// Mitsubishi GX Works2 project: 20150731_final8_test   PLC: Q02/Q02H

PROGRAM MAIN
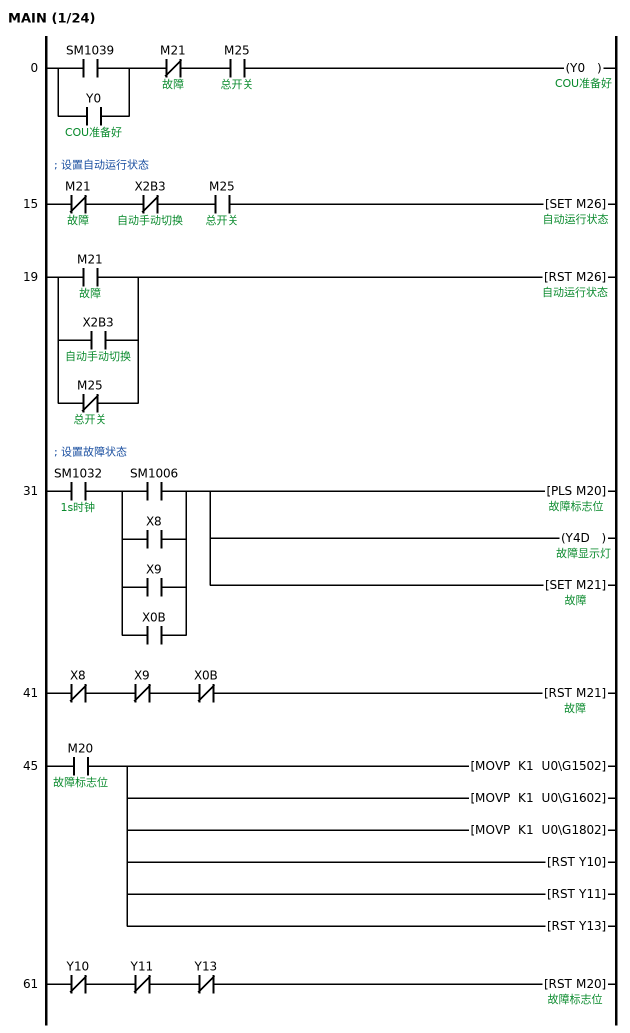
0     LD      SM1039
      OR      Y0  ; COU准备好
      ANI     M21  ; 故障
      AND     M25  ; 总开关
      OUT     Y0  ; COU准备好
; 设置自动运行状态
15    LDI     M21  ; 故障
      ANI     X2B3  ; 自动手动切换
      AND     M25  ; 总开关
      SET     M26  ; 自动运行状态
19    LD      M21  ; 故障
      OR      X2B3  ; 自动手动切换
      ORI     M25  ; 总开关
      RST     M26  ; 自动运行状态
; 设置故障状态
31    LD      SM1032  ; 1s时钟
      LD      SM1006
      OR      X8
      OR      X9
      OR      X0B
      ANB
      PLS     M20  ; 故障标志位
      OUT     Y4D  ; 故障显示灯
      SET     M21  ; 故障
41    LDI     X8
      ANI     X9
      ANI     X0B
      RST     M21  ; 故障
45    LD      M20  ; 故障标志位
      MOVP    K1 U0\G1502
      MOVP    K1 U0\G1602
      MOVP    K1 U0\G1802
      RST     Y10
      RST     Y11
      RST     Y13
61    LDI     Y10
      ANI     Y11
      ANI     Y13
      RST     M20  ; 故障标志位
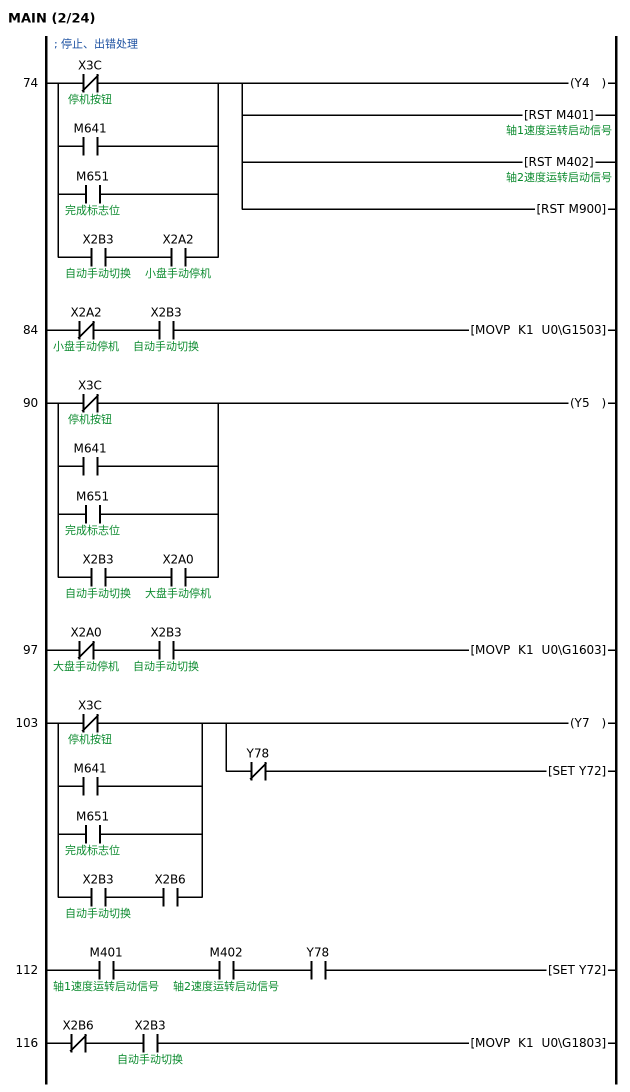
; 停止、出错处理
74    LDI     X3C  ; 停机按钮
      OR      M641
      OR      M651  ; 完成标志位
      LD      X2B3  ; 自动手动切换
      AND     X2A2  ; 小盘手动停机
      ORB
      OUT     Y4
      RST     M401  ; 轴1速度运转启动信号
      RST     M402  ; 轴2速度运转启动信号
      RST     M900
84    LDI     X2A2  ; 小盘手动停机
      AND     X2B3  ; 自动手动切换
      MOVP    K1 U0\G1503
90    LDI     X3C  ; 停机按钮
      OR      M641
      OR      M651  ; 完成标志位
      LD      X2B3  ; 自动手动切换
      AND     X2A0  ; 大盘手动停机
      ORB
      OUT     Y5
97    LDI     X2A0  ; 大盘手动停机
      AND     X2B3  ; 自动手动切换
      MOVP    K1 U0\G1603
103   LDI     X3C  ; 停机按钮
      OR      M641
      OR      M651  ; 完成标志位
      LD      X2B3  ; 自动手动切换
      AND     X2B6
      ORB
      OUT     Y7
      ANI     Y78
      SET     Y72
112   LD      M401  ; 轴1速度运转启动信号
      AND     M402  ; 轴2速度运转启动信号
      AND     Y78
      SET     Y72
116   LDI     X2B6
      AND     X2B3  ; 自动手动切换
      MOVP    K1 U0\G1803
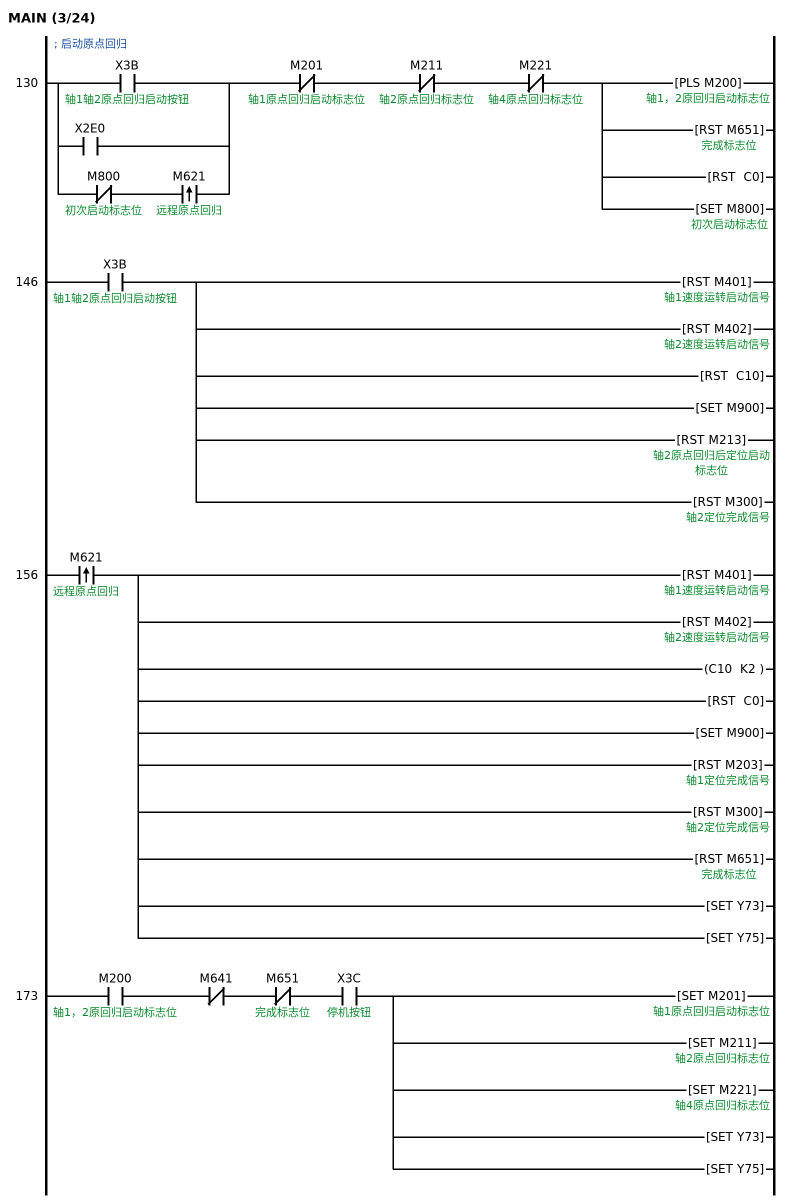
; 启动原点回归
130   LD      X3B  ; 轴1轴2原点回归启动按钮
      OR      X2E0
      LDI     M800  ; 初次启动标志位
      ANDP    M621  ; 远程原点回归
      ORB
      ANI     M201  ; 轴1原点回归启动标志位
      ANI     M211  ; 轴2原点回归标志位
      ANI     M221  ; 轴4原点回归标志位
      PLS     M200  ; 轴1，2原回归启动标志位
      RST     M651  ; 完成标志位
      RST     C0
      SET     M800  ; 初次启动标志位
146   LD      X3B  ; 轴1轴2原点回归启动按钮
      RST     M401  ; 轴1速度运转启动信号
      RST     M402  ; 轴2速度运转启动信号
      RST     C10
      SET     M900
      RST     M213  ; 轴2原点回归后定位启动标志位
      RST     M300  ; 轴2定位完成信号
156   LDP     M621  ; 远程原点回归
      RST     M401  ; 轴1速度运转启动信号
      RST     M402  ; 轴2速度运转启动信号
      OUT     C10 K2
      RST     C0
      SET     M900
      RST     M203  ; 轴1定位完成信号
      RST     M300  ; 轴2定位完成信号
      RST     M651  ; 完成标志位
      SET     Y73
      SET     Y75
173   LD      M200  ; 轴1，2原回归启动标志位
      ANI     M641
      ANI     M651  ; 完成标志位
      AND     X3C  ; 停机按钮
      SET     M201  ; 轴1原点回归启动标志位
      SET     M211  ; 轴2原点回归标志位
      SET     M221  ; 轴4原点回归标志位
      SET     Y73
      SET     Y75
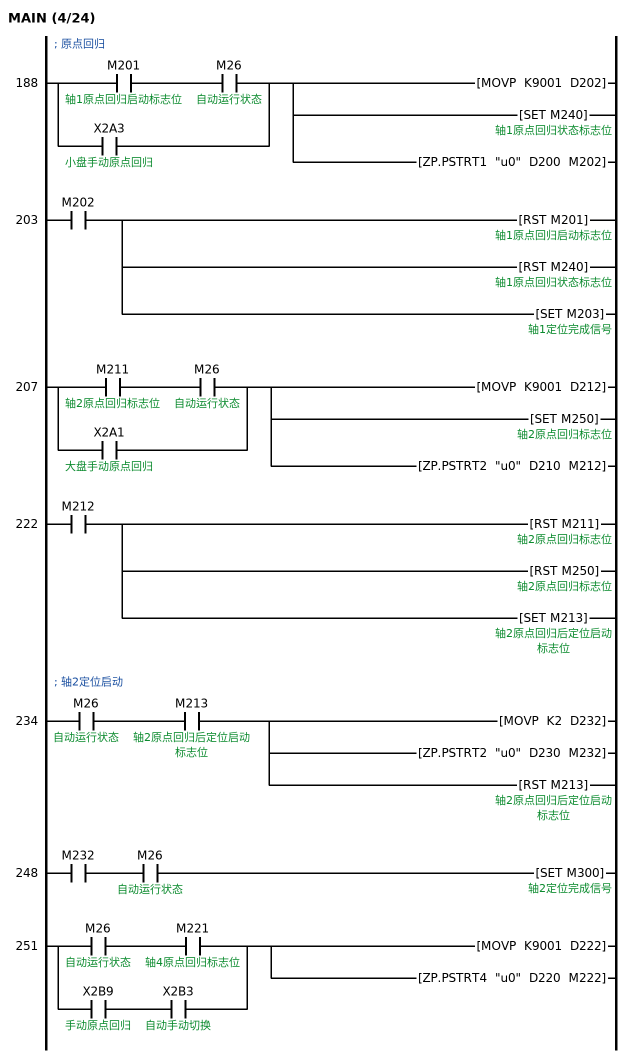
; 原点回归
188   LD      M201  ; 轴1原点回归启动标志位
      AND     M26  ; 自动运行状态
      OR      X2A3  ; 小盘手动原点回归
      MOVP    K9001 D202
      SET     M240  ; 轴1原点回归状态标志位
      ZP.PSTRT1 "u0" D200 M202
203   LD      M202
      RST     M201  ; 轴1原点回归启动标志位
      RST     M240  ; 轴1原点回归状态标志位
      SET     M203  ; 轴1定位完成信号
207   LD      M211  ; 轴2原点回归标志位
      AND     M26  ; 自动运行状态
      OR      X2A1  ; 大盘手动原点回归
      MOVP    K9001 D212
      SET     M250  ; 轴2原点回归标志位
      ZP.PSTRT2 "u0" D210 M212
222   LD      M212
      RST     M211  ; 轴2原点回归标志位
      RST     M250  ; 轴2原点回归标志位
      SET     M213  ; 轴2原点回归后定位启动标志位
; 轴2定位启动
234   LD      M26  ; 自动运行状态
      AND     M213  ; 轴2原点回归后定位启动标志位
      MOVP    K2 D232
      ZP.PSTRT2 "u0" D230 M232
      RST     M213  ; 轴2原点回归后定位启动标志位
248   LD      M232
      AND     M26  ; 自动运行状态
      SET     M300  ; 轴2定位完成信号
251   LD      M26  ; 自动运行状态
      AND     M221  ; 轴4原点回归标志位
      LD      X2B9  ; 手动原点回归
      AND     X2B3  ; 自动手动切换
      ORB
      MOVP    K9001 D222
      ZP.PSTRT4 "u0" D220 M222
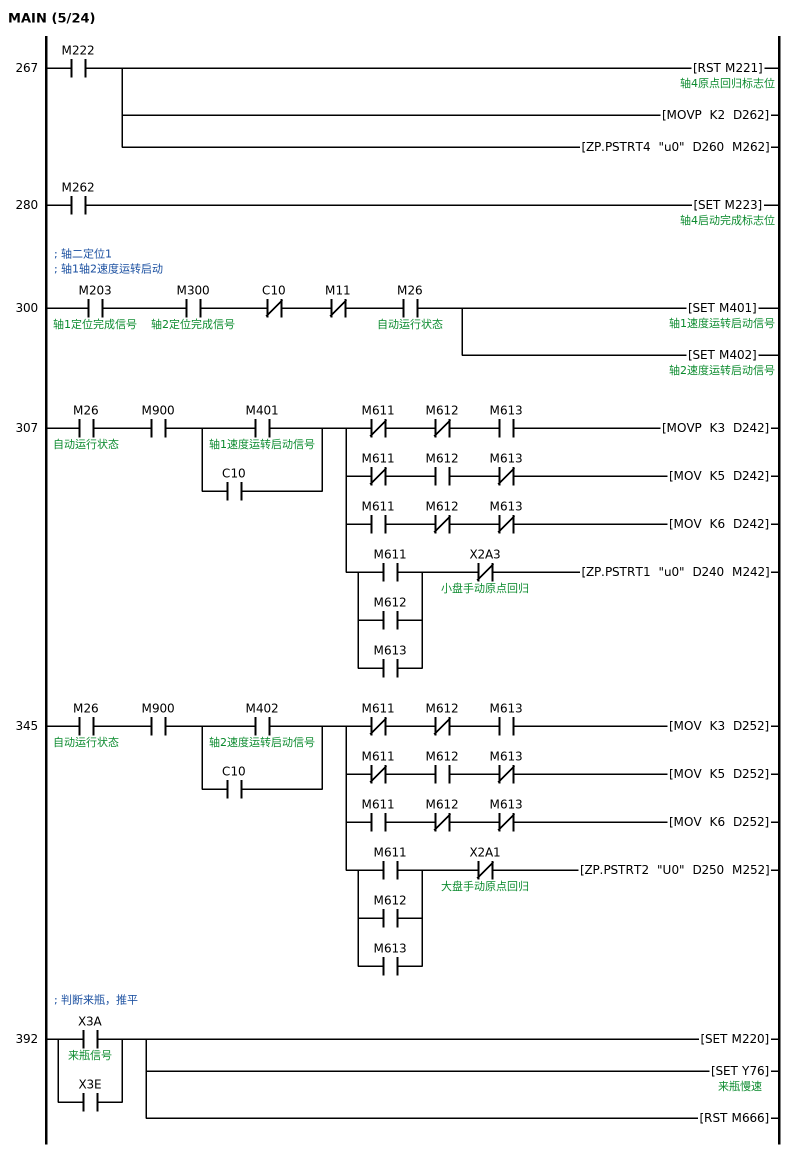
267   LD      M222
      RST     M221  ; 轴4原点回归标志位
      MOVP    K2 D262
      ZP.PSTRT4 "u0" D260 M262
280   LD      M262
      SET     M223  ; 轴4启动完成标志位
; 轴二定位1
; 轴1轴2速度运转启动
300   LD      M203  ; 轴1定位完成信号
      AND     M300  ; 轴2定位完成信号
      ANI     C10
      ANI     M11
      AND     M26  ; 自动运行状态
      SET     M401  ; 轴1速度运转启动信号
      SET     M402  ; 轴2速度运转启动信号
307   LD      M26  ; 自动运行状态
      AND     M900
      LD      M401  ; 轴1速度运转启动信号
      OR      C10
      ANB
      MPS
      ANI     M611
      ANI     M612
      AND     M613
      MOVP    K3 D242
      MRD
      ANI     M611
      AND     M612
      ANI     M613
      MOV     K5 D242
      MRD
      AND     M611
      ANI     M612
      ANI     M613
      MOV     K6 D242
      MPP
      LD      M611
      OR      M612
      OR      M613
      ANB
      ANI     X2A3  ; 小盘手动原点回归
      ZP.PSTRT1 "u0" D240 M242
345   LD      M26  ; 自动运行状态
      AND     M900
      LD      M402  ; 轴2速度运转启动信号
      OR      C10
      ANB
      MPS
      ANI     M611
      ANI     M612
      AND     M613
      MOV     K3 D252
      MRD
      ANI     M611
      AND     M612
      ANI     M613
      MOV     K5 D252
      MRD
      AND     M611
      ANI     M612
      ANI     M613
      MOV     K6 D252
      MPP
      LD      M611
      OR      M612
      OR      M613
      ANB
      ANI     X2A1  ; 大盘手动原点回归
      ZP.PSTRT2 "U0" D250 M252
; 判断来瓶，推平
392   LD      X3A  ; 来瓶信号
      OR      X3E
      SET     M220
      SET     Y76  ; 来瓶慢速
      RST     M666
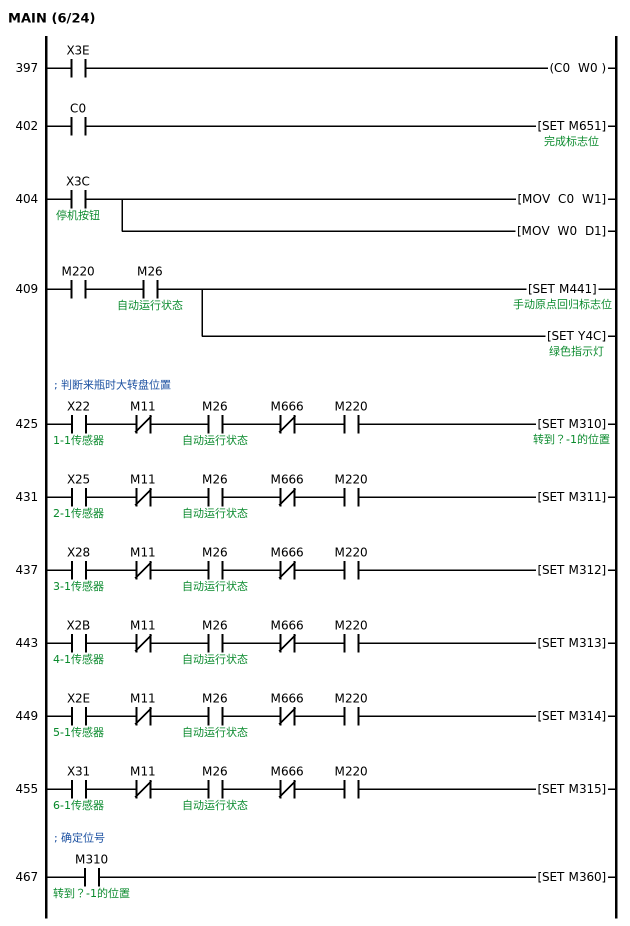
397   LD      X3E
      OUT     C0 W0
402   LD      C0
      SET     M651  ; 完成标志位
404   LD      X3C  ; 停机按钮
      MOV     C0 W1
      MOV     W0 D1
409   LD      M220
      AND     M26  ; 自动运行状态
      SET     M441  ; 手动原点回归标志位
      SET     Y4C  ; 绿色指示灯
; 判断来瓶时大转盘位置
425   LD      X22  ; 1-1传感器
      ANI     M11
      AND     M26  ; 自动运行状态
      ANI     M666
      AND     M220
      SET     M310  ; 转到？-1的位置
431   LD      X25  ; 2-1传感器
      ANI     M11
      AND     M26  ; 自动运行状态
      ANI     M666
      AND     M220
      SET     M311
437   LD      X28  ; 3-1传感器
      ANI     M11
      AND     M26  ; 自动运行状态
      ANI     M666
      AND     M220
      SET     M312
443   LD      X2B  ; 4-1传感器
      ANI     M11
      AND     M26  ; 自动运行状态
      ANI     M666
      AND     M220
      SET     M313
449   LD      X2E  ; 5-1传感器
      ANI     M11
      AND     M26  ; 自动运行状态
      ANI     M666
      AND     M220
      SET     M314
455   LD      X31  ; 6-1传感器
      ANI     M11
      AND     M26  ; 自动运行状态
      ANI     M666
      AND     M220
      SET     M315
; 确定位号
467   LD      M310  ; 转到？-1的位置
      SET     M360
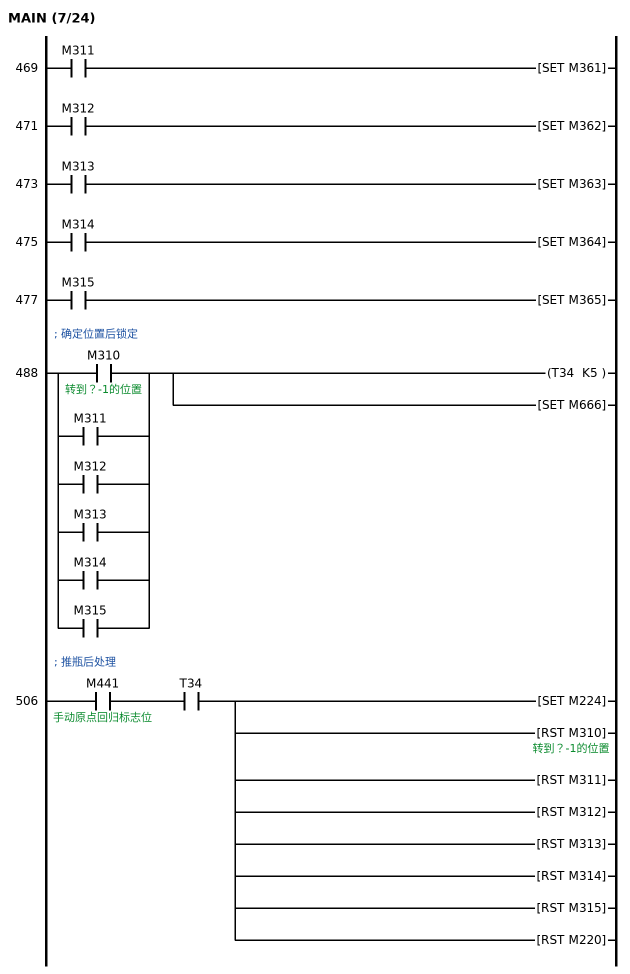
469   LD      M311
      SET     M361
471   LD      M312
      SET     M362
473   LD      M313
      SET     M363
475   LD      M314
      SET     M364
477   LD      M315
      SET     M365
; 确定位置后锁定
488   LD      M310  ; 转到？-1的位置
      OR      M311
      OR      M312
      OR      M313
      OR      M314
      OR      M315
      OUT     T34 K5
      SET     M666
; 推瓶后处理
506   LD      M441  ; 手动原点回归标志位
      AND     T34
      SET     M224
      RST     M310  ; 转到？-1的位置
      RST     M311
      RST     M312
      RST     M313
      RST     M314
      RST     M315
      RST     M220
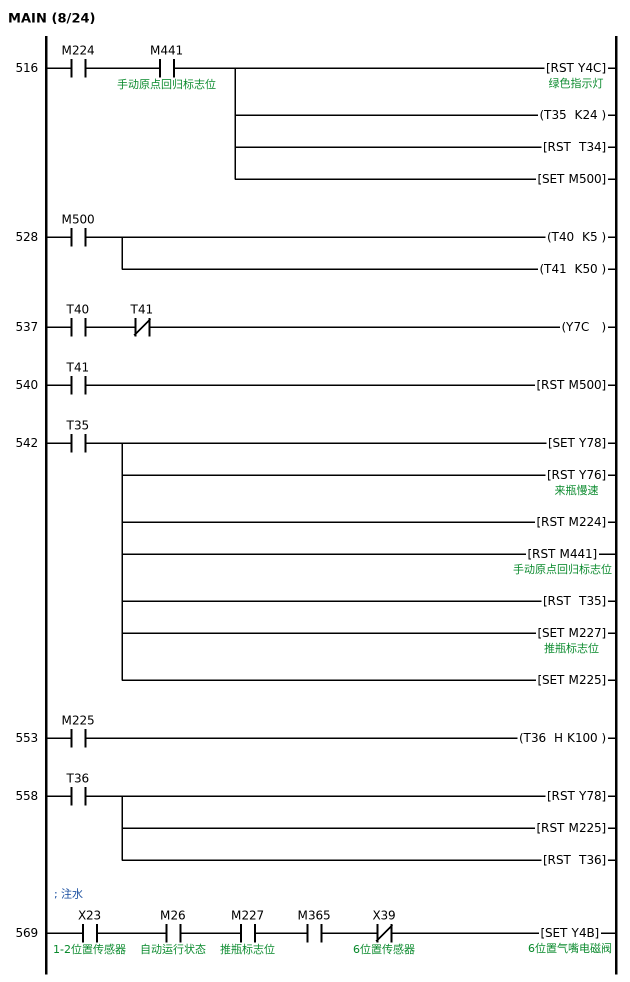
516   LD      M224
      AND     M441  ; 手动原点回归标志位
      RST     Y4C  ; 绿色指示灯
      OUT     T35 K24
      RST     T34
      SET     M500
528   LD      M500
      OUT     T40 K5
      OUT     T41 K50
537   LD      T40
      ANI     T41
      OUT     Y7C
540   LD      T41
      RST     M500
542   LD      T35
      SET     Y78
      RST     Y76  ; 来瓶慢速
      RST     M224
      RST     M441  ; 手动原点回归标志位
      RST     T35
      SET     M227  ; 推瓶标志位
      SET     M225
553   LD      M225
      OUTH    T36 K100
558   LD      T36
      RST     Y78
      RST     M225
      RST     T36
; 注水
569   LD      X23  ; 1-2位置传感器
      AND     M26  ; 自动运行状态
      AND     M227  ; 推瓶标志位
      AND     M365
      ANI     X39  ; 6位置传感器
      SET     Y4B  ; 6位置气嘴电磁阀
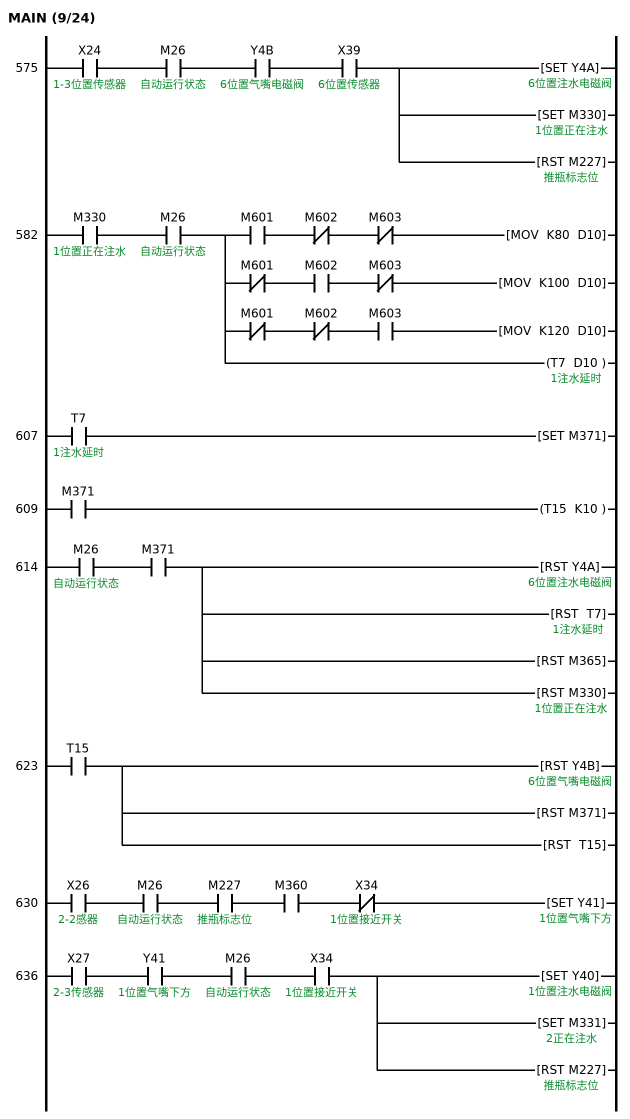
575   LD      X24  ; 1-3位置传感器
      AND     M26  ; 自动运行状态
      AND     Y4B  ; 6位置气嘴电磁阀
      AND     X39  ; 6位置传感器
      SET     Y4A  ; 6位置注水电磁阀
      SET     M330  ; 1位置正在注水
      RST     M227  ; 推瓶标志位
582   LD      M330  ; 1位置正在注水
      AND     M26  ; 自动运行状态
      MPS
      AND     M601
      ANI     M602
      ANI     M603
      MOV     K80 D10
      MRD
      ANI     M601
      AND     M602
      ANI     M603
      MOV     K100 D10
      MRD
      ANI     M601
      ANI     M602
      AND     M603
      MOV     K120 D10
      MPP
      OUT     T7 D10  ; 1注水延时
607   LD      T7  ; 1注水延时
      SET     M371
609   LD      M371
      OUT     T15 K10
614   LD      M26  ; 自动运行状态
      AND     M371
      RST     Y4A  ; 6位置注水电磁阀
      RST     T7  ; 1注水延时
      RST     M365
      RST     M330  ; 1位置正在注水
623   LD      T15
      RST     Y4B  ; 6位置气嘴电磁阀
      RST     M371
      RST     T15
630   LD      X26  ; 2-2感器
      AND     M26  ; 自动运行状态
      AND     M227  ; 推瓶标志位
      AND     M360
      ANI     X34  ; 1位置接近开关
      SET     Y41  ; 1位置气嘴下方
636   LD      X27  ; 2-3传感器
      AND     Y41  ; 1位置气嘴下方
      AND     M26  ; 自动运行状态
      AND     X34  ; 1位置接近开关
      SET     Y40  ; 1位置注水电磁阀
      SET     M331  ; 2正在注水
      RST     M227  ; 推瓶标志位
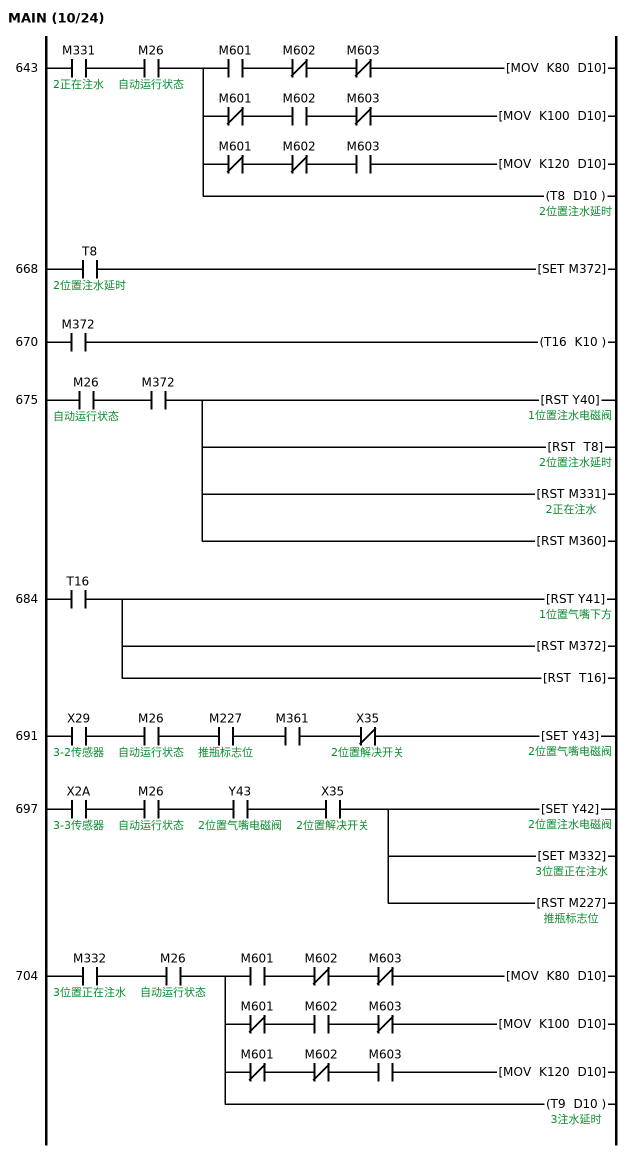
643   LD      M331  ; 2正在注水
      AND     M26  ; 自动运行状态
      MPS
      AND     M601
      ANI     M602
      ANI     M603
      MOV     K80 D10
      MRD
      ANI     M601
      AND     M602
      ANI     M603
      MOV     K100 D10
      MRD
      ANI     M601
      ANI     M602
      AND     M603
      MOV     K120 D10
      MPP
      OUT     T8 D10  ; 2位置注水延时
668   LD      T8  ; 2位置注水延时
      SET     M372
670   LD      M372
      OUT     T16 K10
675   LD      M26  ; 自动运行状态
      AND     M372
      RST     Y40  ; 1位置注水电磁阀
      RST     T8  ; 2位置注水延时
      RST     M331  ; 2正在注水
      RST     M360
684   LD      T16
      RST     Y41  ; 1位置气嘴下方
      RST     M372
      RST     T16
691   LD      X29  ; 3-2传感器
      AND     M26  ; 自动运行状态
      AND     M227  ; 推瓶标志位
      AND     M361
      ANI     X35  ; 2位置解决开关
      SET     Y43  ; 2位置气嘴电磁阀
697   LD      X2A  ; 3-3传感器
      AND     M26  ; 自动运行状态
      AND     Y43  ; 2位置气嘴电磁阀
      AND     X35  ; 2位置解决开关
      SET     Y42  ; 2位置注水电磁阀
      SET     M332  ; 3位置正在注水
      RST     M227  ; 推瓶标志位
704   LD      M332  ; 3位置正在注水
      AND     M26  ; 自动运行状态
      MPS
      AND     M601
      ANI     M602
      ANI     M603
      MOV     K80 D10
      MRD
      ANI     M601
      AND     M602
      ANI     M603
      MOV     K100 D10
      MRD
      ANI     M601
      ANI     M602
      AND     M603
      MOV     K120 D10
      MPP
      OUT     T9 D10  ; 3注水延时
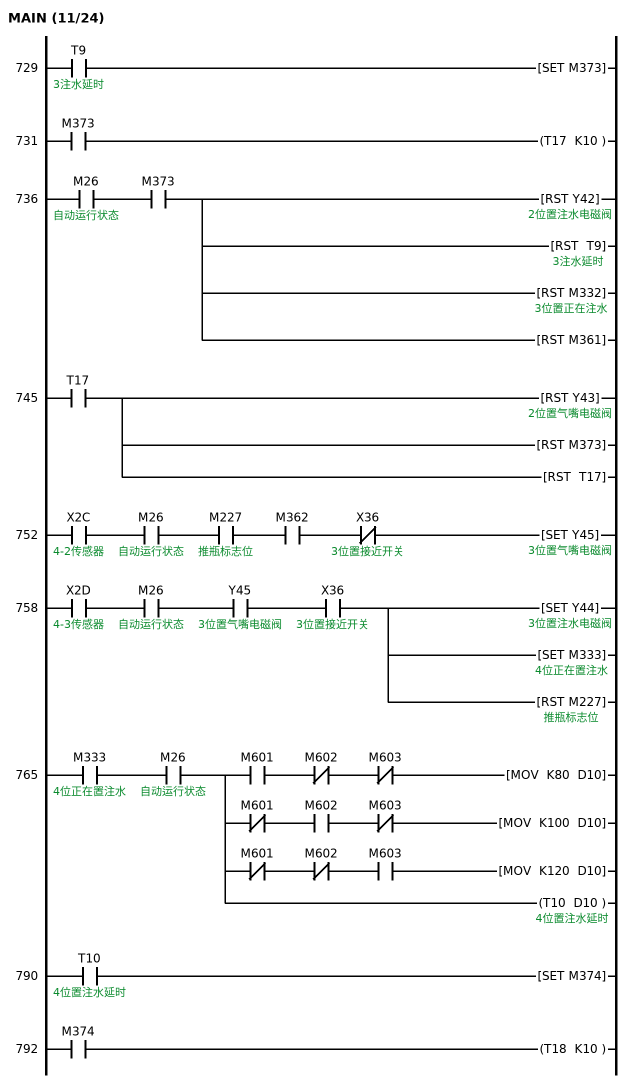
729   LD      T9  ; 3注水延时
      SET     M373
731   LD      M373
      OUT     T17 K10
736   LD      M26  ; 自动运行状态
      AND     M373
      RST     Y42  ; 2位置注水电磁阀
      RST     T9  ; 3注水延时
      RST     M332  ; 3位置正在注水
      RST     M361
745   LD      T17
      RST     Y43  ; 2位置气嘴电磁阀
      RST     M373
      RST     T17
752   LD      X2C  ; 4-2传感器
      AND     M26  ; 自动运行状态
      AND     M227  ; 推瓶标志位
      AND     M362
      ANI     X36  ; 3位置接近开关
      SET     Y45  ; 3位置气嘴电磁阀
758   LD      X2D  ; 4-3传感器
      AND     M26  ; 自动运行状态
      AND     Y45  ; 3位置气嘴电磁阀
      AND     X36  ; 3位置接近开关
      SET     Y44  ; 3位置注水电磁阀
      SET     M333  ; 4位正在置注水
      RST     M227  ; 推瓶标志位
765   LD      M333  ; 4位正在置注水
      AND     M26  ; 自动运行状态
      MPS
      AND     M601
      ANI     M602
      ANI     M603
      MOV     K80 D10
      MRD
      ANI     M601
      AND     M602
      ANI     M603
      MOV     K100 D10
      MRD
      ANI     M601
      ANI     M602
      AND     M603
      MOV     K120 D10
      MPP
      OUT     T10 D10  ; 4位置注水延时
790   LD      T10  ; 4位置注水延时
      SET     M374
792   LD      M374
      OUT     T18 K10
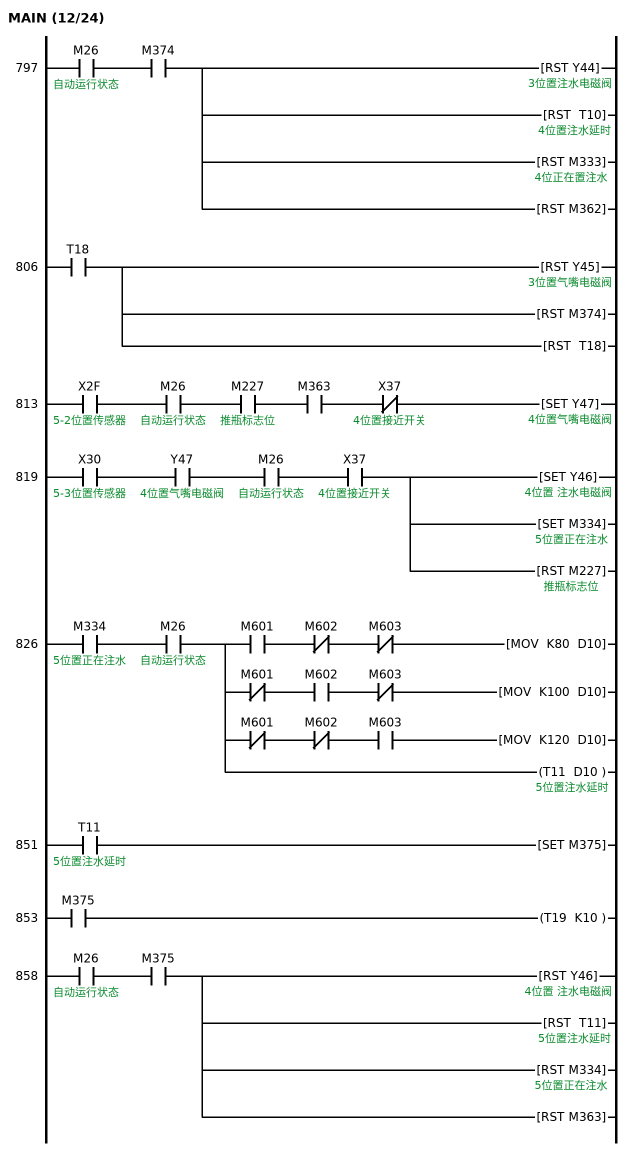
797   LD      M26  ; 自动运行状态
      AND     M374
      RST     Y44  ; 3位置注水电磁阀
      RST     T10  ; 4位置注水延时
      RST     M333  ; 4位正在置注水
      RST     M362
806   LD      T18
      RST     Y45  ; 3位置气嘴电磁阀
      RST     M374
      RST     T18
813   LD      X2F  ; 5-2位置传感器
      AND     M26  ; 自动运行状态
      AND     M227  ; 推瓶标志位
      AND     M363
      ANI     X37  ; 4位置接近开关
      SET     Y47  ; 4位置气嘴电磁阀
819   LD      X30  ; 5-3位置传感器
      AND     Y47  ; 4位置气嘴电磁阀
      AND     M26  ; 自动运行状态
      AND     X37  ; 4位置接近开关
      SET     Y46  ; 4位置 注水电磁阀
      SET     M334  ; 5位置正在注水
      RST     M227  ; 推瓶标志位
826   LD      M334  ; 5位置正在注水
      AND     M26  ; 自动运行状态
      MPS
      AND     M601
      ANI     M602
      ANI     M603
      MOV     K80 D10
      MRD
      ANI     M601
      AND     M602
      ANI     M603
      MOV     K100 D10
      MRD
      ANI     M601
      ANI     M602
      AND     M603
      MOV     K120 D10
      MPP
      OUT     T11 D10  ; 5位置注水延时
851   LD      T11  ; 5位置注水延时
      SET     M375
853   LD      M375
      OUT     T19 K10
858   LD      M26  ; 自动运行状态
      AND     M375
      RST     Y46  ; 4位置 注水电磁阀
      RST     T11  ; 5位置注水延时
      RST     M334  ; 5位置正在注水
      RST     M363
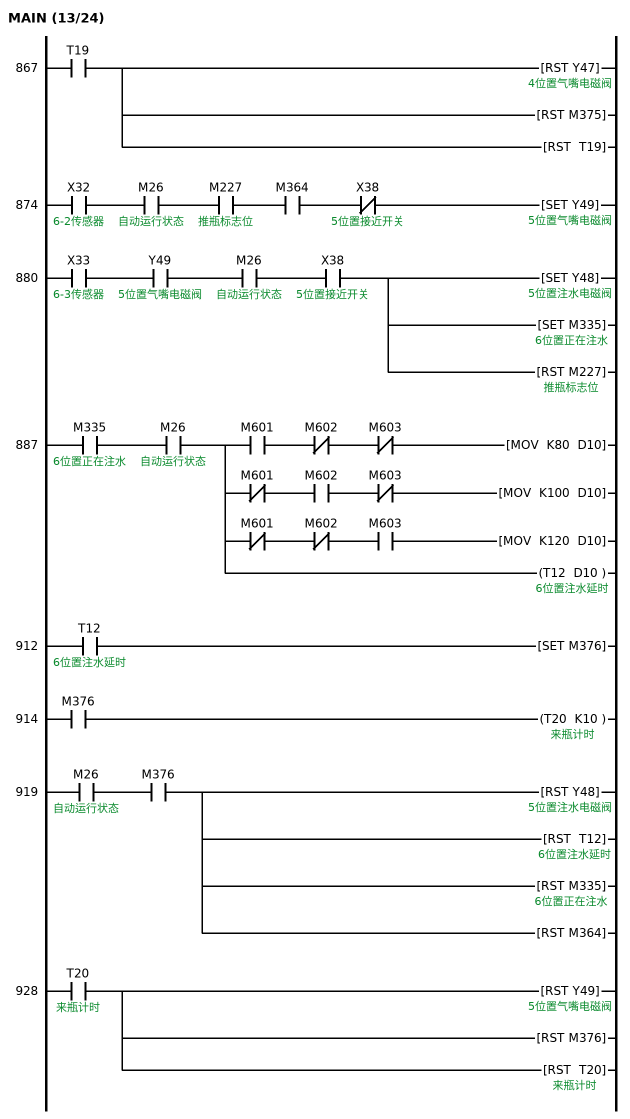
867   LD      T19
      RST     Y47  ; 4位置气嘴电磁阀
      RST     M375
      RST     T19
874   LD      X32  ; 6-2传感器
      AND     M26  ; 自动运行状态
      AND     M227  ; 推瓶标志位
      AND     M364
      ANI     X38  ; 5位置接近开关
      SET     Y49  ; 5位置气嘴电磁阀
880   LD      X33  ; 6-3传感器
      AND     Y49  ; 5位置气嘴电磁阀
      AND     M26  ; 自动运行状态
      AND     X38  ; 5位置接近开关
      SET     Y48  ; 5位置注水电磁阀
      SET     M335  ; 6位置正在注水
      RST     M227  ; 推瓶标志位
887   LD      M335  ; 6位置正在注水
      AND     M26  ; 自动运行状态
      MPS
      AND     M601
      ANI     M602
      ANI     M603
      MOV     K80 D10
      MRD
      ANI     M601
      AND     M602
      ANI     M603
      MOV     K100 D10
      MRD
      ANI     M601
      ANI     M602
      AND     M603
      MOV     K120 D10
      MPP
      OUT     T12 D10  ; 6位置注水延时
912   LD      T12  ; 6位置注水延时
      SET     M376
914   LD      M376
      OUT     T20 K10  ; 来瓶计时
919   LD      M26  ; 自动运行状态
      AND     M376
      RST     Y48  ; 5位置注水电磁阀
      RST     T12  ; 6位置注水延时
      RST     M335  ; 6位置正在注水
      RST     M364
928   LD      T20  ; 来瓶计时
      RST     Y49  ; 5位置气嘴电磁阀
      RST     M376
      RST     T20  ; 来瓶计时
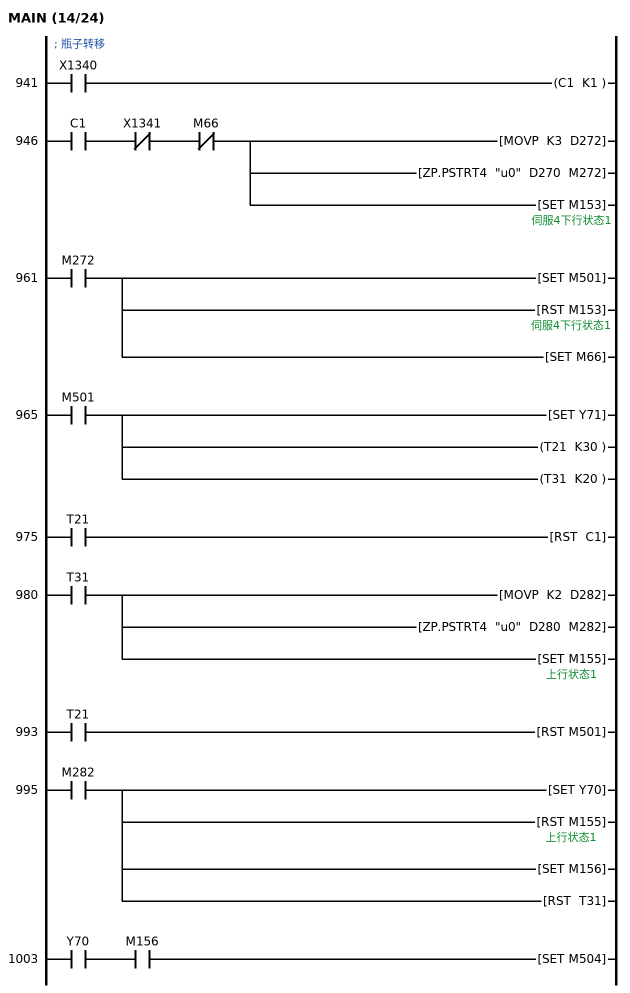
; 瓶子转移
941   LD      X1340
      OUT     C1 K1
946   LD      C1
      ANI     X1341
      ANI     M66
      MOVP    K3 D272
      ZP.PSTRT4 "u0" D270 M272
      SET     M153  ; 伺服4下行状态1
961   LD      M272
      SET     M501
      RST     M153  ; 伺服4下行状态1
      SET     M66
965   LD      M501
      SET     Y71
      OUT     T21 K30
      OUT     T31 K20
975   LD      T21
      RST     C1
980   LD      T31
      MOVP    K2 D282
      ZP.PSTRT4 "u0" D280 M282
      SET     M155  ; 上行状态1
993   LD      T21
      RST     M501
995   LD      M282
      SET     Y70
      RST     M155  ; 上行状态1
      SET     M156
      RST     T31
1003  LD      Y70
      AND     M156
      SET     M504
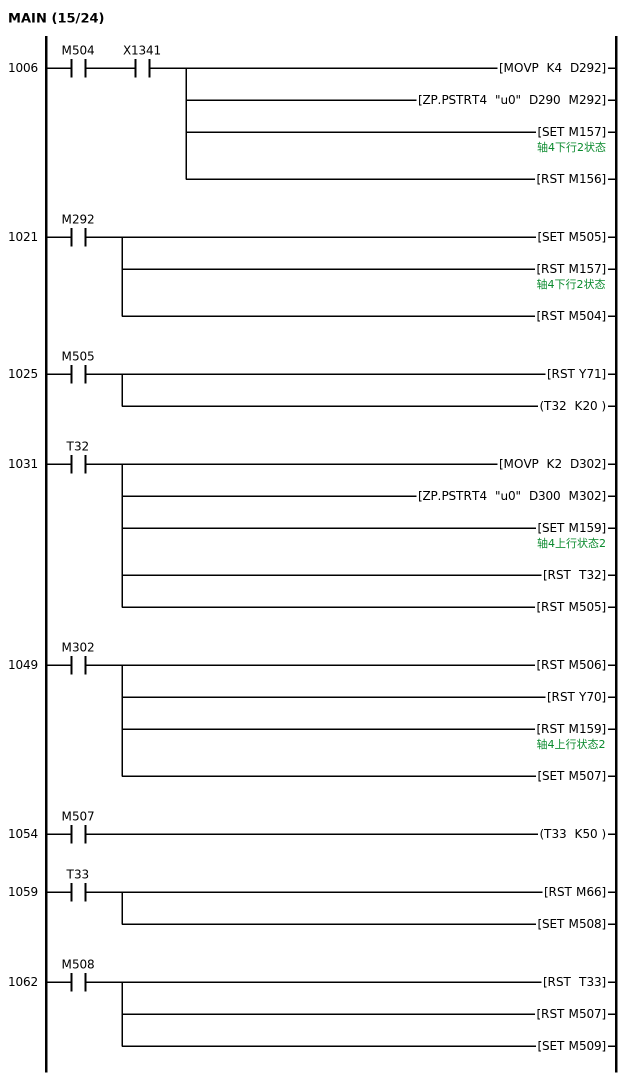
1006  LD      M504
      AND     X1341
      MOVP    K4 D292
      ZP.PSTRT4 "u0" D290 M292
      SET     M157  ; 轴4下行2状态
      RST     M156
1021  LD      M292
      SET     M505
      RST     M157  ; 轴4下行2状态
      RST     M504
1025  LD      M505
      RST     Y71
      OUT     T32 K20
1031  LD      T32
      MOVP    K2 D302
      ZP.PSTRT4 "u0" D300 M302
      SET     M159  ; 轴4上行状态2
      RST     T32
      RST     M505
1049  LD      M302
      RST     M506
      RST     Y70
      RST     M159  ; 轴4上行状态2
      SET     M507
1054  LD      M507
      OUT     T33 K50
1059  LD      T33
      RST     M66
      SET     M508
1062  LD      M508
      RST     T33
      RST     M507
      SET     M509
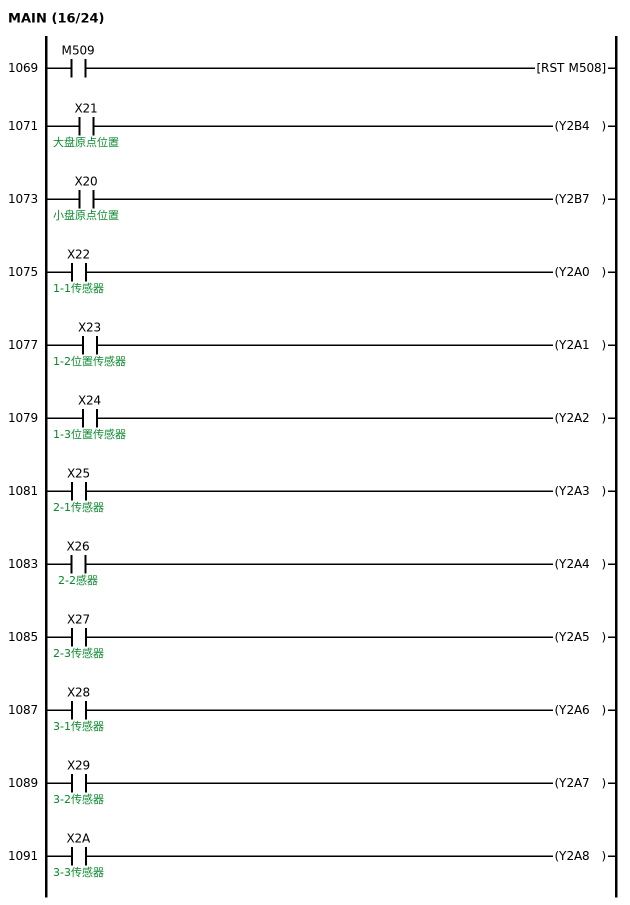
1069  LD      M509
      RST     M508
1071  LD      X21  ; 大盘原点位置
      OUT     Y2B4
1073  LD      X20  ; 小盘原点位置
      OUT     Y2B7
1075  LD      X22  ; 1-1传感器
      OUT     Y2A0
1077  LD      X23  ; 1-2位置传感器
      OUT     Y2A1
1079  LD      X24  ; 1-3位置传感器
      OUT     Y2A2
1081  LD      X25  ; 2-1传感器
      OUT     Y2A3
1083  LD      X26  ; 2-2感器
      OUT     Y2A4
1085  LD      X27  ; 2-3传感器
      OUT     Y2A5
1087  LD      X28  ; 3-1传感器
      OUT     Y2A6
1089  LD      X29  ; 3-2传感器
      OUT     Y2A7
1091  LD      X2A  ; 3-3传感器
      OUT     Y2A8
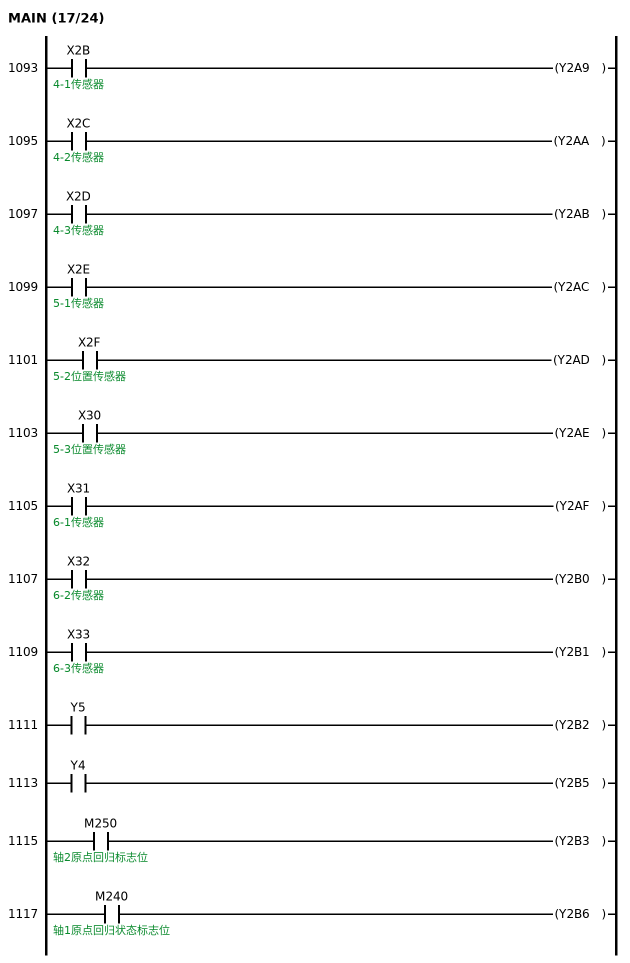
1093  LD      X2B  ; 4-1传感器
      OUT     Y2A9
1095  LD      X2C  ; 4-2传感器
      OUT     Y2AA
1097  LD      X2D  ; 4-3传感器
      OUT     Y2AB
1099  LD      X2E  ; 5-1传感器
      OUT     Y2AC
1101  LD      X2F  ; 5-2位置传感器
      OUT     Y2AD
1103  LD      X30  ; 5-3位置传感器
      OUT     Y2AE
1105  LD      X31  ; 6-1传感器
      OUT     Y2AF
1107  LD      X32  ; 6-2传感器
      OUT     Y2B0
1109  LD      X33  ; 6-3传感器
      OUT     Y2B1
1111  LD      Y5
      OUT     Y2B2
1113  LD      Y4
      OUT     Y2B5
1115  LD      M250  ; 轴2原点回归标志位
      OUT     Y2B3
1117  LD      M240  ; 轴1原点回归状态标志位
      OUT     Y2B6
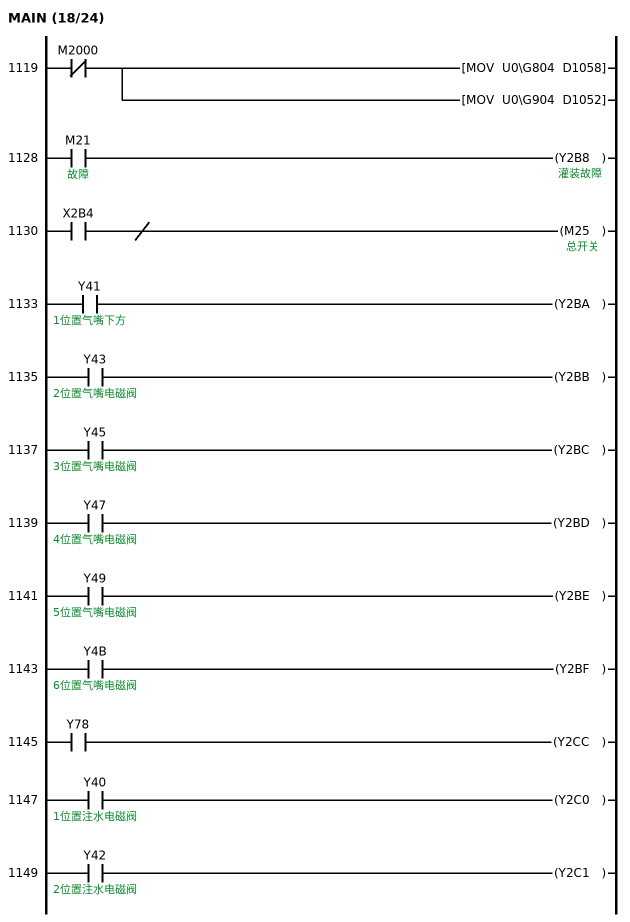
1119  LDI     M2000
      MOV     U0\G804 D1058
      MOV     U0\G904 D1052
1128  LD      M21  ; 故障
      OUT     Y2B8  ; 灌装故障
1130  LD      X2B4
      INV
      OUT     M25  ; 总开关
1133  LD      Y41  ; 1位置气嘴下方
      OUT     Y2BA
1135  LD      Y43  ; 2位置气嘴电磁阀
      OUT     Y2BB
1137  LD      Y45  ; 3位置气嘴电磁阀
      OUT     Y2BC
1139  LD      Y47  ; 4位置气嘴电磁阀
      OUT     Y2BD
1141  LD      Y49  ; 5位置气嘴电磁阀
      OUT     Y2BE
1143  LD      Y4B  ; 6位置气嘴电磁阀
      OUT     Y2BF
1145  LD      Y78
      OUT     Y2CC
1147  LD      Y40  ; 1位置注水电磁阀
      OUT     Y2C0
1149  LD      Y42  ; 2位置注水电磁阀
      OUT     Y2C1
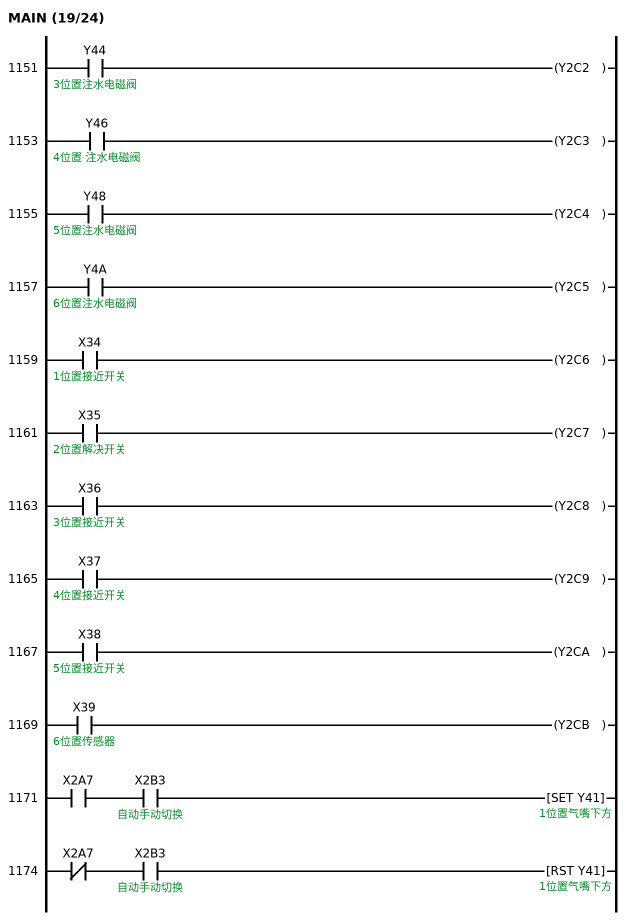
1151  LD      Y44  ; 3位置注水电磁阀
      OUT     Y2C2
1153  LD      Y46  ; 4位置 注水电磁阀
      OUT     Y2C3
1155  LD      Y48  ; 5位置注水电磁阀
      OUT     Y2C4
1157  LD      Y4A  ; 6位置注水电磁阀
      OUT     Y2C5
1159  LD      X34  ; 1位置接近开关
      OUT     Y2C6
1161  LD      X35  ; 2位置解决开关
      OUT     Y2C7
1163  LD      X36  ; 3位置接近开关
      OUT     Y2C8
1165  LD      X37  ; 4位置接近开关
      OUT     Y2C9
1167  LD      X38  ; 5位置接近开关
      OUT     Y2CA
1169  LD      X39  ; 6位置传感器
      OUT     Y2CB
1171  LD      X2A7
      AND     X2B3  ; 自动手动切换
      SET     Y41  ; 1位置气嘴下方
1174  LDI     X2A7
      AND     X2B3  ; 自动手动切换
      RST     Y41  ; 1位置气嘴下方
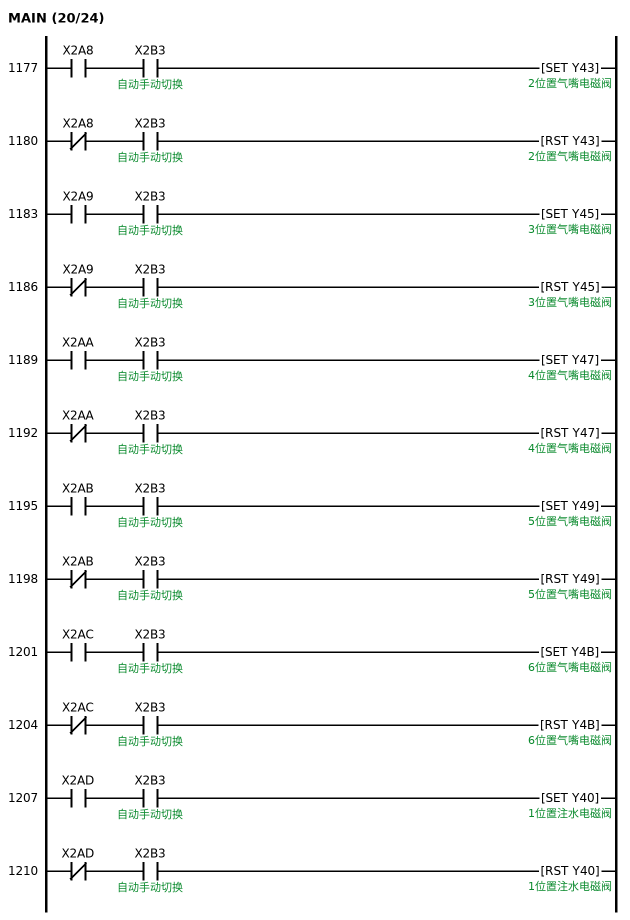
1177  LD      X2A8
      AND     X2B3  ; 自动手动切换
      SET     Y43  ; 2位置气嘴电磁阀
1180  LDI     X2A8
      AND     X2B3  ; 自动手动切换
      RST     Y43  ; 2位置气嘴电磁阀
1183  LD      X2A9
      AND     X2B3  ; 自动手动切换
      SET     Y45  ; 3位置气嘴电磁阀
1186  LDI     X2A9
      AND     X2B3  ; 自动手动切换
      RST     Y45  ; 3位置气嘴电磁阀
1189  LD      X2AA
      AND     X2B3  ; 自动手动切换
      SET     Y47  ; 4位置气嘴电磁阀
1192  LDI     X2AA
      AND     X2B3  ; 自动手动切换
      RST     Y47  ; 4位置气嘴电磁阀
1195  LD      X2AB
      AND     X2B3  ; 自动手动切换
      SET     Y49  ; 5位置气嘴电磁阀
1198  LDI     X2AB
      AND     X2B3  ; 自动手动切换
      RST     Y49  ; 5位置气嘴电磁阀
1201  LD      X2AC
      AND     X2B3  ; 自动手动切换
      SET     Y4B  ; 6位置气嘴电磁阀
1204  LDI     X2AC
      AND     X2B3  ; 自动手动切换
      RST     Y4B  ; 6位置气嘴电磁阀
1207  LD      X2AD
      AND     X2B3  ; 自动手动切换
      SET     Y40  ; 1位置注水电磁阀
1210  LDI     X2AD
      AND     X2B3  ; 自动手动切换
      RST     Y40  ; 1位置注水电磁阀
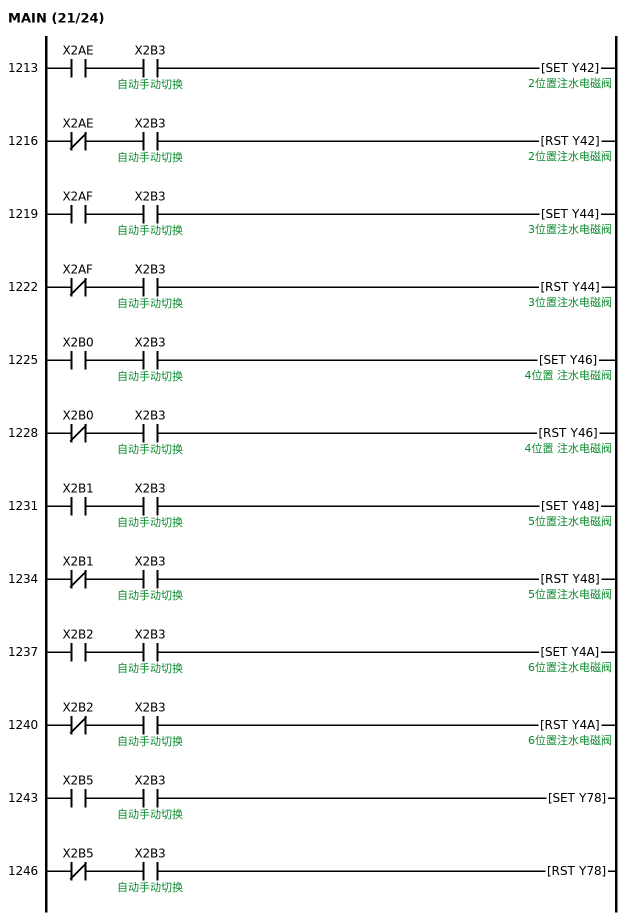
1213  LD      X2AE
      AND     X2B3  ; 自动手动切换
      SET     Y42  ; 2位置注水电磁阀
1216  LDI     X2AE
      AND     X2B3  ; 自动手动切换
      RST     Y42  ; 2位置注水电磁阀
1219  LD      X2AF
      AND     X2B3  ; 自动手动切换
      SET     Y44  ; 3位置注水电磁阀
1222  LDI     X2AF
      AND     X2B3  ; 自动手动切换
      RST     Y44  ; 3位置注水电磁阀
1225  LD      X2B0
      AND     X2B3  ; 自动手动切换
      SET     Y46  ; 4位置 注水电磁阀
1228  LDI     X2B0
      AND     X2B3  ; 自动手动切换
      RST     Y46  ; 4位置 注水电磁阀
1231  LD      X2B1
      AND     X2B3  ; 自动手动切换
      SET     Y48  ; 5位置注水电磁阀
1234  LDI     X2B1
      AND     X2B3  ; 自动手动切换
      RST     Y48  ; 5位置注水电磁阀
1237  LD      X2B2
      AND     X2B3  ; 自动手动切换
      SET     Y4A  ; 6位置注水电磁阀
1240  LDI     X2B2
      AND     X2B3  ; 自动手动切换
      RST     Y4A  ; 6位置注水电磁阀
1243  LD      X2B5
      AND     X2B3  ; 自动手动切换
      SET     Y78
1246  LDI     X2B5
      AND     X2B3  ; 自动手动切换
      RST     Y78
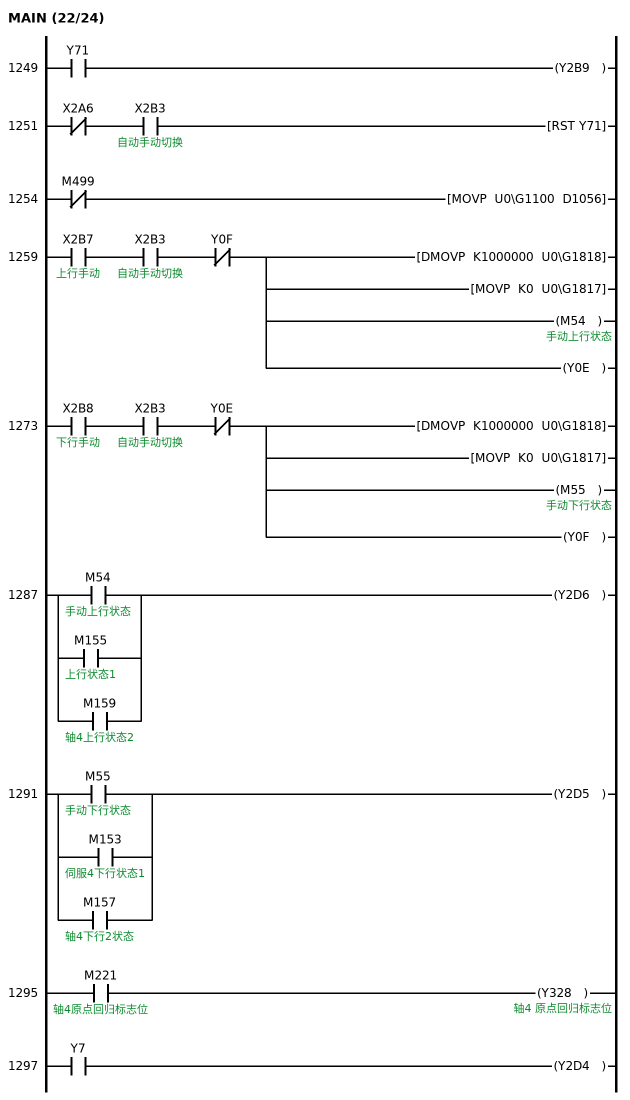
1249  LD      Y71
      OUT     Y2B9
1251  LDI     X2A6
      AND     X2B3  ; 自动手动切换
      RST     Y71
1254  LDI     M499
      MOVP    U0\G1100 D1056
1259  LD      X2B7  ; 上行手动
      AND     X2B3  ; 自动手动切换
      ANI     Y0F
      DMOVP   K1000000 U0\G1818
      MOVP    K0 U0\G1817
      OUT     M54  ; 手动上行状态
      OUT     Y0E
1273  LD      X2B8  ; 下行手动
      AND     X2B3  ; 自动手动切换
      ANI     Y0E
      DMOVP   K1000000 U0\G1818
      MOVP    K0 U0\G1817
      OUT     M55  ; 手动下行状态
      OUT     Y0F
1287  LD      M54  ; 手动上行状态
      OR      M155  ; 上行状态1
      OR      M159  ; 轴4上行状态2
      OUT     Y2D6
1291  LD      M55  ; 手动下行状态
      OR      M153  ; 伺服4下行状态1
      OR      M157  ; 轴4下行2状态
      OUT     Y2D5
1295  LD      M221  ; 轴4原点回归标志位
      OUT     Y328  ; 轴4 原点回归标志位
1297  LD      Y7
      OUT     Y2D4
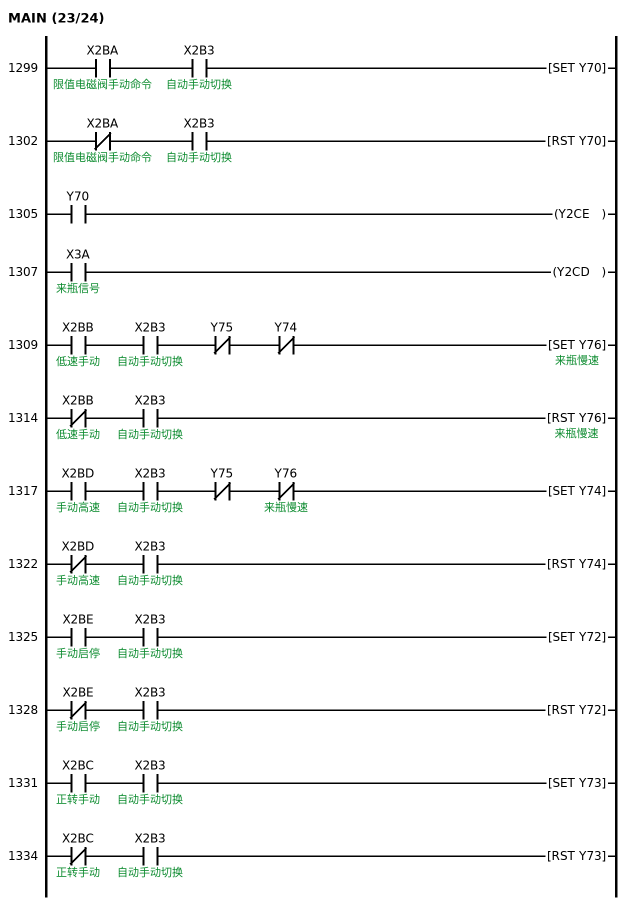
1299  LD      X2BA  ; 限值电磁阀手动命令
      AND     X2B3  ; 自动手动切换
      SET     Y70
1302  LDI     X2BA  ; 限值电磁阀手动命令
      AND     X2B3  ; 自动手动切换
      RST     Y70
1305  LD      Y70
      OUT     Y2CE
1307  LD      X3A  ; 来瓶信号
      OUT     Y2CD
1309  LD      X2BB  ; 低速手动
      AND     X2B3  ; 自动手动切换
      ANI     Y75
      ANI     Y74
      SET     Y76  ; 来瓶慢速
1314  LDI     X2BB  ; 低速手动
      AND     X2B3  ; 自动手动切换
      RST     Y76  ; 来瓶慢速
1317  LD      X2BD  ; 手动高速
      AND     X2B3  ; 自动手动切换
      ANI     Y75
      ANI     Y76  ; 来瓶慢速
      SET     Y74
1322  LDI     X2BD  ; 手动高速
      AND     X2B3  ; 自动手动切换
      RST     Y74
1325  LD      X2BE  ; 手动启停
      AND     X2B3  ; 自动手动切换
      SET     Y72
1328  LDI     X2BE  ; 手动启停
      AND     X2B3  ; 自动手动切换
      RST     Y72
1331  LD      X2BC  ; 正转手动
      AND     X2B3  ; 自动手动切换
      SET     Y73
1334  LDI     X2BC  ; 正转手动
      AND     X2B3  ; 自动手动切换
      RST     Y73
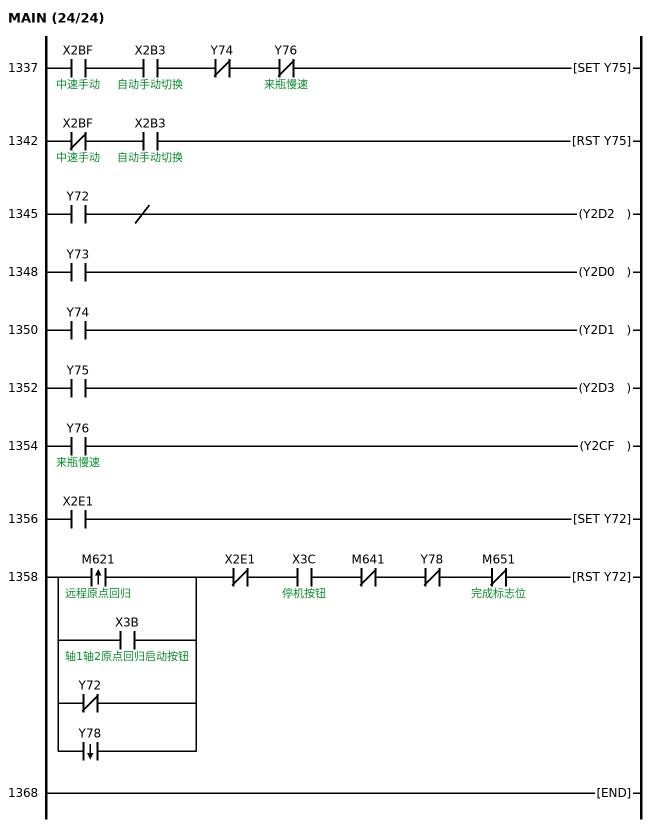
1337  LD      X2BF  ; 中速手动
      AND     X2B3  ; 自动手动切换
      ANI     Y74
      ANI     Y76  ; 来瓶慢速
      SET     Y75
1342  LDI     X2BF  ; 中速手动
      AND     X2B3  ; 自动手动切换
      RST     Y75
1345  LD      Y72
      INV
      OUT     Y2D2
1348  LD      Y73
      OUT     Y2D0
1350  LD      Y74
      OUT     Y2D1
1352  LD      Y75
      OUT     Y2D3
1354  LD      Y76  ; 来瓶慢速
      OUT     Y2CF
1356  LD      X2E1
      SET     Y72
1358  LDP     M621  ; 远程原点回归
      OR      X3B  ; 轴1轴2原点回归启动按钮
      ORI     Y72
      ORF     Y78
      ANI     X2E1
      AND     X3C  ; 停机按钮
      ANI     M641
      ANI     Y78
      ANI     M651  ; 完成标志位
      RST     Y72
1368  END
END_PROGRAM

// device comments not shown above
X2A4  ; 出瓶信号1
X2A5  ; 出瓶信号2
Y50  ; 机械手旋转电磁阀
Y51  ; 气爪电磁阀
Y52  ; 启动
Y53  ; 正转
Y54  ; 高速
Y55  ; 中速
Y56  ; 低速
M31  ; 瓶进入1-1位置
M32  ; 瓶进入2-1位置
M33  ; 瓶进入3-1位置
M34  ; 瓶进入4-1位置
M35  ; 瓶进入5-1位置
M36  ; 瓶进入6-1位置
M41  ; 1位瓶正在处理
M42  ; 2位瓶正在处理
M43  ; 3位置瓶正在处理
M44  ; 4位瓶正在处理
M45  ; 5位置瓶正在处理
M46  ; 6位瓶正在处理
M160  ; 在待机位
M260  ; 中速状态位
M261  ; 交流高速状态
M301  ; 轴1原点回归完成信号
M420  ; 等待？-2的动作
M421  ; 1-2位置准备动作
M422  ; 2-2位置准备动作
M423  ; 3-2位置准备动作
M424  ; 4-2位置准备动作
M425  ; 5-2位置准备动作
M426  ; 6-2位置准备动作
M431  ; 有瓶等待被推入
M631  ; 远程启动信号
T1  ; 推瓶动作持续1S后结束
